// TIA Portal V15.1 export
// export: Created 2020-12-07T09:03:51.9968235Z, ExportSetting WithDefaults, WithReadOnly, DisplayName Totally Integrated Automation Portal, DisplayVersion V15.1 Update 4, DisplayName TIA Portal Openness, DisplayVersion V15.1, DisplayName SINAMICS Startdrive Advanced, DisplayVersion V15.1 Update3, DisplayName SINAMICS Startdrive G110M, G120, G120C, G120D, G120P, DisplayVersion V15.1 Update3, DisplayName SINAMICS Startdrive G130, G150, S120, S150, SINAMICS MV, S210, DisplayVersion V15.1 Update3, DisplayName STEP 7 Professional, DisplayVersion V15.1 Update 4, DisplayName STEP 7 Safety, DisplayVersion V15.1, DisplayName WinCC Professional, DisplayVersion V15.1 Update 4
VAR_GLOBAL   // PLC tag table "OUTPUT_ST_A"
   "Y1A/BA" AT %Q2000.0 : Bool;
   "Y1B/BA" AT %Q2000.1 : Bool;
   "Y2A/BA" AT %Q2000.2 : Bool;
   "Y2B/BA" AT %Q2000.3 : Bool;
   "Y3A/BA" AT %Q2000.4 : Bool;
   "Y3B/BA" AT %Q2000.5 : Bool;
   "Y4A/BA" AT %Q2000.6 : Bool;
   "Y4B/BA" AT %Q2000.7 : Bool;
   "Y5A/BA" AT %Q2001.0 : Bool;
   "Y5B/BA" AT %Q2001.1 : Bool;
   "Y6A/BA" AT %Q2001.2 : Bool;
   "Y6B/BA" AT %Q2001.3 : Bool;
   "Y7A/BA" AT %Q2001.4 : Bool;
   "Y7B/BA" AT %Q2001.5 : Bool;
   "Y8A/BA" AT %Q2001.6 : Bool;
   "Y8B/BA" AT %Q2001.7 : Bool;
   "Y9A/BA" AT %Q2002.0 : Bool;
   "Y9B/BA" AT %Q2002.1 : Bool;
   "Y10A/BA" AT %Q2002.2 : Bool;
   "Y10B/BA" AT %Q2002.3 : Bool;
   "Y11A/BA" AT %Q2002.4 : Bool;
   "Y11B/BA" AT %Q2002.5 : Bool;
   "Y12A/BA" AT %Q2002.6 : Bool;
   "Y12B/BA" AT %Q2002.7 : Bool;
   "Y13A/BA" AT %Q2003.0 : Bool;
   "Y13B/BA" AT %Q2003.1 : Bool;
   "Y14A/BA" AT %Q2003.2 : Bool;
   "Y14B/BA" AT %Q2003.3 : Bool;
   "Y15A/BA" AT %Q2003.4 : Bool;
   "EV_SPARE_30/BA" AT %Q2003.5 : Bool;
   "EV_SPARE_31/BA" AT %Q2003.6 : Bool;
   "EV_SPARE_32/BA" AT %Q2003.7 : Bool;
   "Y17A/BA" AT %Q2100.0 : Bool;
   "Y17B/BA" AT %Q2100.1 : Bool;
   "Y18A/BA" AT %Q2100.2 : Bool;
   "Y18B/BA" AT %Q2100.3 : Bool;
   "Y19A/BA" AT %Q2100.4 : Bool;
   "Y19B/BA" AT %Q2100.5 : Bool;
   "Y20A/BA" AT %Q2100.6 : Bool;
   "Y20B/BA" AT %Q2100.7 : Bool;
   "Y21A/BA" AT %Q2101.0 : Bool;
   "Y21B/BA" AT %Q2101.1 : Bool;
   "Y22A/BA" AT %Q2101.2 : Bool;
   "Y22B/BA" AT %Q2101.3 : Bool;
   "Y23A/BA" AT %Q2101.4 : Bool;
   "Y23B/BA" AT %Q2101.5 : Bool;
   "Y24A/BA" AT %Q2101.6 : Bool;
   "Y24B/BA" AT %Q2101.7 : Bool;
   "Y25A/BA" AT %Q2102.0 : Bool;
   "Y25B/BA" AT %Q2102.1 : Bool;
   "Y26A/BA" AT %Q2102.2 : Bool;
   "Y26B/BA" AT %Q2102.3 : Bool;
   "Y27A/BA" AT %Q2102.4 : Bool;
   "Y27B/BA" AT %Q2102.5 : Bool;
   "Y28A/BA" AT %Q2102.6 : Bool;
   "Y28B/BA" AT %Q2102.7 : Bool;
   "Y29A/BA" AT %Q2103.0 : Bool;
   "EV_SPARE_58/BA" AT %Q2103.1 : Bool;
   "EV_SPARE_59/BA" AT %Q2103.2 : Bool;
   "EV_SPARE_60/BA" AT %Q2103.3 : Bool;
   "EV_SPARE_61/BA" AT %Q2103.4 : Bool;
   "EV_SPARE_62/BA" AT %Q2103.5 : Bool;
   "EV_SPARE_63/BA" AT %Q2103.6 : Bool;
   "EV_SPARE_64/BA" AT %Q2103.7 : Bool;
   "RESET_LASER/BA" AT %Q12.0 : Bool;
   "POWER_AZ4/BA" AT %Q12.1 : Bool;
   "POWER_AZ5/BA" AT %Q12.2 : Bool;
   "POWER_AZ6/BA" AT %Q12.3 : Bool;
   "POWER_AZ7/BA" AT %Q12.4 : Bool;
   "POWER_AZ8/BA" AT %Q12.5 : Bool;
   "POWER_AZ9/BA" AT %Q12.6 : Bool;
   "POWER_AZ10/BA" AT %Q12.7 : Bool;
   "RESET_AZ27/BA" AT %Q13.1 : Bool;
   "DRIVEON_AZ27/BA" AT %Q13.0 : Bool;
   "POWER_AZ12/BA" AT %Q13.2 : Bool;
   "POWER_AZ13/BA" AT %Q13.3 : Bool;
   "POWER_AZ15/BA" AT %Q13.4 : Bool;
   "POWER_AZ17/BA" AT %Q13.5 : Bool;
   "POWER_AZ19/BA" AT %Q13.6 : Bool;
   "POWER_AZ21/BA" AT %Q13.7 : Bool;
   "POWER_AZ23/BA" AT %Q14.0 : Bool;
   "POWER_AZ25/BA" AT %Q14.1 : Bool;
   "POWER_AZ26/BA" AT %Q14.2 : Bool;
   "OIL_MOTOR/BA" AT %Q14.3 : Bool;
   "POWER_AZ27/BA" AT %Q14.4 : Bool;
   "EMG_REQUEST/BA" AT %Q14.5 : Bool;
   "Y_ENDCAP_LOCK_SX/BA" AT %Q14.7 : Bool;
   "Y_ENDCAP_LOCK_DX/BA" AT %Q14.6 : Bool;
   "Y_OIL_LOOP/BA" AT %Q15.0 : Bool;
   "Y_SEEGER_LOCK_SX/BA" AT %Q15.2 : Bool;
   "Y_SEEGER_LOCK_DX/BA" AT %Q15.1 : Bool;
   "SEM_EC_B0/BA" AT %QB2010 : Byte;
   "SEM_EC_B1/BA" AT %QB2011 : Byte;
   "SEM_EC_B2/BA" AT %QB2012 : Byte;
   "ANALOG_AZ27/BA" AT %QW18 : Word;
   "AZ15/BA_HomingFC" AT %Q16.6 : Bool;
   "AZ12/BA_HomingFC" AT %Q16.7 : Bool;
   "Y_GLUE_1A_SX/BA" AT %Q15.3 : Bool;
   "Y_GLUE_2A_SX/BA" AT %Q15.7 : Bool;
   "Y_GLUE_1A_DX/BA" AT %Q15.5 : Bool;
   "Y_GLUE_2A_DX/BA" AT %Q16.0 : Bool;
   "Y_GLUE_1B_SX/BA" AT %Q15.4 : Bool;
   "Y_GLUE_1B_DX/BA" AT %Q15.6 : Bool;
END_VAR
